Fanuc KAREL source: RGET_SREGCMT.kl

PROGRAM T
%NOLOCKGROUP
VAR
 v0 : STRING[40]
 v1 : INTEGER
 v2 : STRING[40]
 v3 : INTEGER
BEGIN
 RGET_SREGCMT(v0, v1, v2, v3)
END T
